// TIA Portal V19 export
TYPE "C403_VAR_LVE_TYPIC"
   STRUCT
      BSC { ExternalAccessible := 'False'; ExternalVisible := 'False'; ExternalWritable := 'False'} : USInt;   // Beschikbaarheid
      STS_NEG { ExternalAccessible := 'False'; ExternalVisible := 'False'; ExternalWritable := 'False'} : USInt;   // Spookrijder gedetecteerd
      OBS { ExternalAccessible := 'False'; ExternalVisible := 'False'; ExternalWritable := 'False'} : USInt;   // Observeerbaarheid
      SIG_AV01 { ExternalAccessible := 'False'; ExternalVisible := 'False'; ExternalWritable := 'False'} : USInt;   // Signalering Stilstand gedetecteerd actief
      SIG_AV02 { ExternalAccessible := 'False'; ExternalVisible := 'False'; ExternalWritable := 'False'} : USInt;   // Signalering Snelheidsonderschrijding actief
      POS { ExternalAccessible := 'False'; ExternalVisible := 'False'; ExternalWritable := 'False'} : Bool;   // Positie van het detectiepunt
   END_STRUCT;
END_TYPE
